{attribute 'qualified_only'}
//{attribute 'strict'}
{attribute 'to_string'}
TYPE E_NCI_STATE :
(
  NULL,
  INIT,
  IDLE,
  RESET,
  LOAD_PROG,
  FEED_TABLE,
  BUILD_GROUP,
  CLEAR_GROUP,

  START         := 10,
  STOP,
  STO_STOP,
  RESTART_STEP_ON,

  M_FUNC_QUIT   := 20,

  READ_R_PARA   := 30,
  WRITE_R_PARA  := 40

)UINT;
END_TYPE

(* stored: Version 1.1.0.1
   DUT E_NCI_STATE: Id {5aed9498-2ef8-4009-9f3f-53565340a806} *)
